(* LS Electric XG5000 project: 241007_TON,TOF 사용 *)
(* PLC LSPLC *)
(* module base 0 slot 0: 입력 모듈:XGI-D22A/B (DC 24V 입력, 16점 (전류소스 싱크공용/ 전류소스 입력)) *)
(* module base 0 slot 1: 출력 모듈:XGQ-RY2A/B (릴레이 출력, 16점 (2A용, Varistor 없음/Varistor 부착)) *)

PROGRAM NewProgram (* task: 스캔 프로그램 *)
VAR
    T1 : TON;
    T2 : TOF;
    T4 : TP;
    time02 : TIME := T#3s;
    time04 : TIME := T#2s; (* 2초 *)
    time5s : TIME := T#5s; (* 5초 *)
    램프_1 AT %QX0.1.0 : BOOL;
    램프_2 AT %QX0.1.1 : BOOL;
    램프_3 AT %QX0.1.2 : BOOL;
    램프_4 AT %QX0.1.3 : BOOL;
    스위치_T1 AT %IX0.0.0 : BOOL;
    스위치_T2 AT %IX0.0.1 : BOOL;
    스위치_T3 AT %IX0.0.2 : BOOL;
    스위치_T4 AT %IX0.0.3 : BOOL;
END_VAR

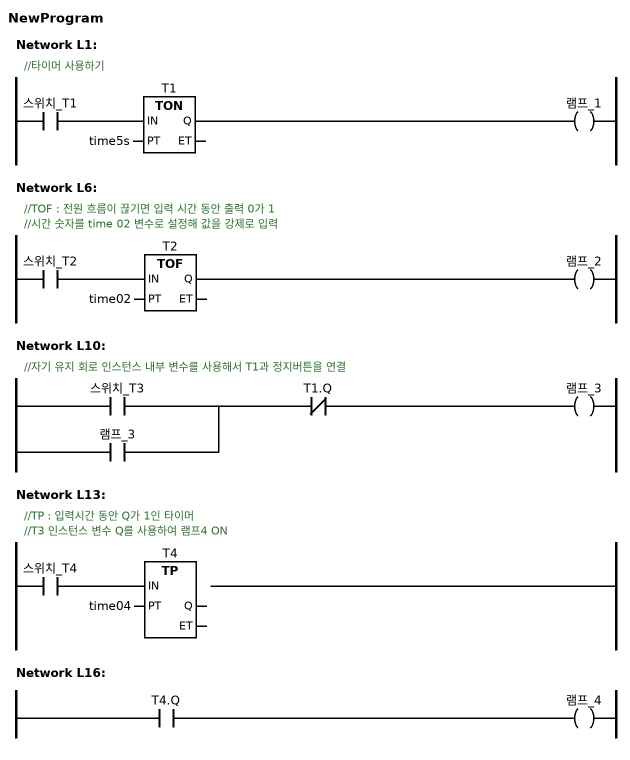
(* //타이머 사용하기 *)
(* Rung L1 *)
T1(IN := 스위치_T1, PT := time5s);
램프_1 := T1.Q;
(* //TOF : 전원 흐름이 끊기면 입력 시간 동안 출력 0가 1 *)
(* //시간 숫자를 time 02 변수로 설정해 값을 강제로 입력 *)
(* Rung L6 *)
T2(IN := 스위치_T2, PT := time02);
램프_2 := T2.Q;
(* //자기 유지 회로 인스턴스 내부 변수를 사용해서 T1과 정지버튼을 연결 *)
(* Rung L10 *)
램프_3 := (스위치_T3 OR 램프_3) AND NOT T1.Q;
(* //TP : 입력시간 동안 Q가 1인 타이머 / //T3 인스턴스 변수 Q를 사용하여 램프4 ON *)
(* Rung L13 *)
T4(IN := 스위치_T4, PT := time04);
(* Rung L16 *)
램프_4 := T4.Q;
END_PROGRAM